FUNCTION Buffer_Layout_Set_String_Array : UINT
VAR_INPUT
END_VAR
VAR
END_VAR

END_FUNCTION

(* stored: Version 1.1.0.1, ProductVersion 3.1.4024.10
   POU Buffer_Layout_Set_String_Array: Id {cf0ddbea-b9b2-44af-9e2f-56dfedf2d1b5}, SpecialFunc None *)
